INTERFACE ITF_BaseLogger

METHOD PUBLIC AddItem : INT
VAR_INPUT
	itfItem				: ITF_BaseLogger_Item;
END_VAR
END_METHOD

METHOD PUBLIC GetNumerOfReportsIntheSystem : UINT
VAR_INPUT
END_VAR
END_METHOD

METHOD PUBLIC ReportEvent : BOOL
VAR_INPUT
	stEvent					: ST_BaseEvents_RowInQueue;
END_VAR
END_METHOD

METHOD PUBLIC SetNumerOfReportsIntheSystem
VAR_INPUT
	uiValue		: UINT;
END_VAR
END_METHOD

END_INTERFACE

(* stored: Version 1.1.0.1
   Itf ITF_BaseLogger: Id {dde1500f-ba43-0973-2072-39e8d4239f74}
   Method AddItem: Id {0dd39ff2-6376-09aa-21a8-e3d343fc09ac}
   Method GetNumerOfReportsIntheSystem: Id {9aacd584-e7e1-09b4-05c5-c971f6539be5}
   Method ReportEvent: Id {bf8e154d-88a6-07c9-1886-c0d273a4c7f4}
   Method SetNumerOfReportsIntheSystem: Id {660e0beb-bd67-0d21-3c2e-25250f190eba} *)
